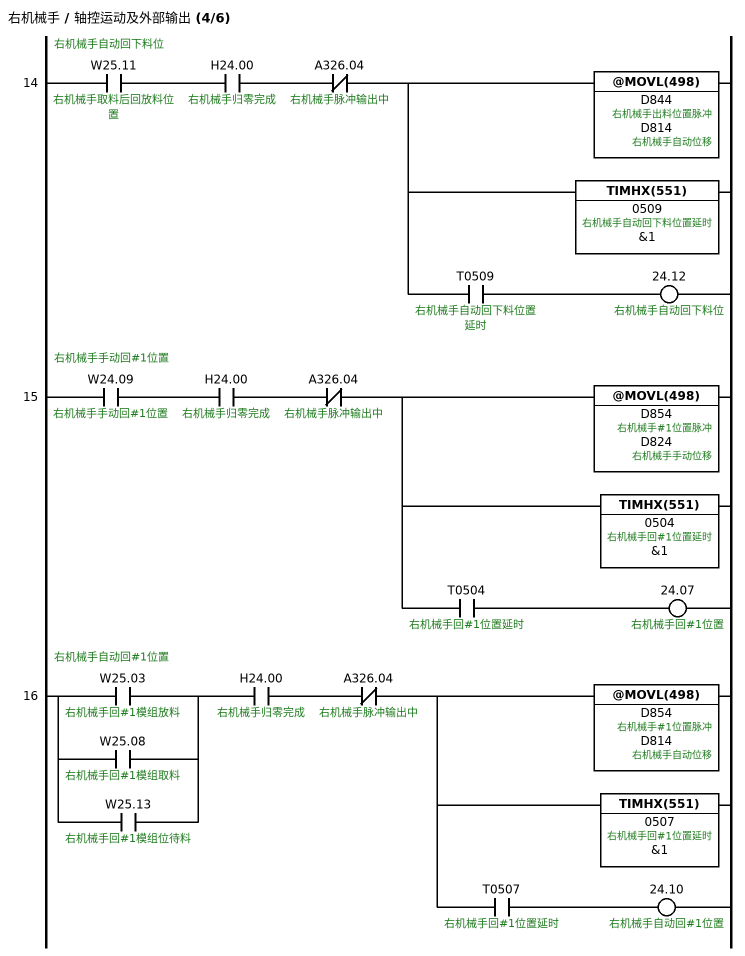
; [picture p185: 右机械手 / 轴控运动及外部输出, rungs 14-16]
; rung 14: 右机械手自动回下料位
LD W25.11  ; 右机械手取料后回放料位置
AND H24.00  ; 右机械手归零完成
ANDNOT A326.04  ; 右机械手脉冲输出中
@MOVL(498) D844 D814  ; 右机械手出料位置脉冲, 右机械手自动位移
TIMHX(551) 0509 &1  ; 右机械手自动回下料位置延时
AND T0509  ; 右机械手自动回下料位置延时
OUT 24.12  ; 右机械手自动回下料位
; rung 15: 右机械手手动回#1位置
LD W24.09  ; 右机械手手动回#1位置
AND H24.00  ; 右机械手归零完成
ANDNOT A326.04  ; 右机械手脉冲输出中
@MOVL(498) D854 D824  ; 右机械手#1位置脉冲, 右机械手手动位移
TIMHX(551) 0504 &1  ; 右机械手回#1位置延时
AND T0504  ; 右机械手回#1位置延时
OUT 24.07  ; 右机械手回#1位置
; rung 16: 右机械手自动回#1位置
LD W25.03  ; 右机械手回#1模组放料
OR W25.08  ; 右机械手回#1模组取料
OR W25.13  ; 右机械手回#1模组位待料
AND H24.00  ; 右机械手归零完成
ANDNOT A326.04  ; 右机械手脉冲输出中
@MOVL(498) D854 D814  ; 右机械手#1位置脉冲, 右机械手自动位移
TIMHX(551) 0507 &1  ; 右机械手回#1位置延时
AND T0507  ; 右机械手回#1位置延时
OUT 24.10  ; 右机械手自动回#1位置

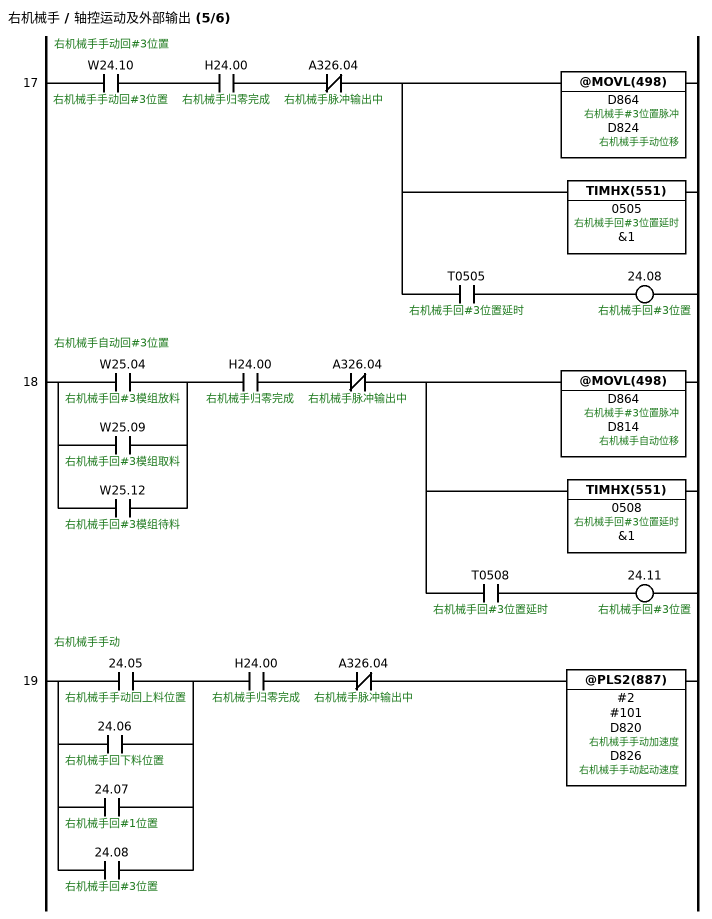
; rung 17: 右机械手手动回#3位置
LD W24.10  ; 右机械手手动回#3位置
AND H24.00  ; 右机械手归零完成
ANDNOT A326.04  ; 右机械手脉冲输出中
@MOVL(498) D864 D824  ; 右机械手#3位置脉冲, 右机械手手动位移
TIMHX(551) 0505 &1  ; 右机械手回#3位置延时
AND T0505  ; 右机械手回#3位置延时
OUT 24.08  ; 右机械手回#3位置
; rung 18: 右机械手自动回#3位置
LD W25.04  ; 右机械手回#3模组放料
OR W25.09  ; 右机械手回#3模组取料
OR W25.12  ; 右机械手回#3模组待料
AND H24.00  ; 右机械手归零完成
ANDNOT A326.04  ; 右机械手脉冲输出中
@MOVL(498) D864 D814  ; 右机械手#3位置脉冲, 右机械手自动位移
TIMHX(551) 0508 &1  ; 右机械手回#3位置延时
AND T0508  ; 右机械手回#3位置延时
OUT 24.11  ; 右机械手回#3位置
; rung 19: 右机械手手动
LD 24.05  ; 右机械手手动回上料位置
OR 24.06  ; 右机械手回下料位置
OR 24.07  ; 右机械手回#1位置
OR 24.08  ; 右机械手回#3位置
AND H24.00  ; 右机械手归零完成
ANDNOT A326.04  ; 右机械手脉冲输出中
@PLS2(887) #2 #101 D820 D826  ; 右机械手手动加速度, 右机械手手动起动速度

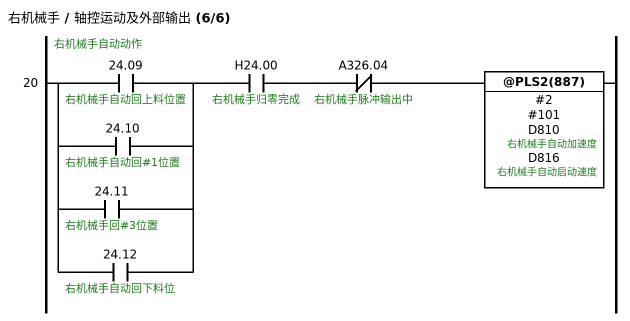
; rung 20: 右机械手自动动作
LD 24.09  ; 右机械手自动回上料位置
OR 24.10  ; 右机械手自动回#1位置
OR 24.11  ; 右机械手回#3位置
OR 24.12  ; 右机械手自动回下料位
AND H24.00  ; 右机械手归零完成
ANDNOT A326.04  ; 右机械手脉冲输出中
@PLS2(887) #2 #101 D810 D816  ; 右机械手自动加速度, 右机械手自动启动速度

### Section 自动报警

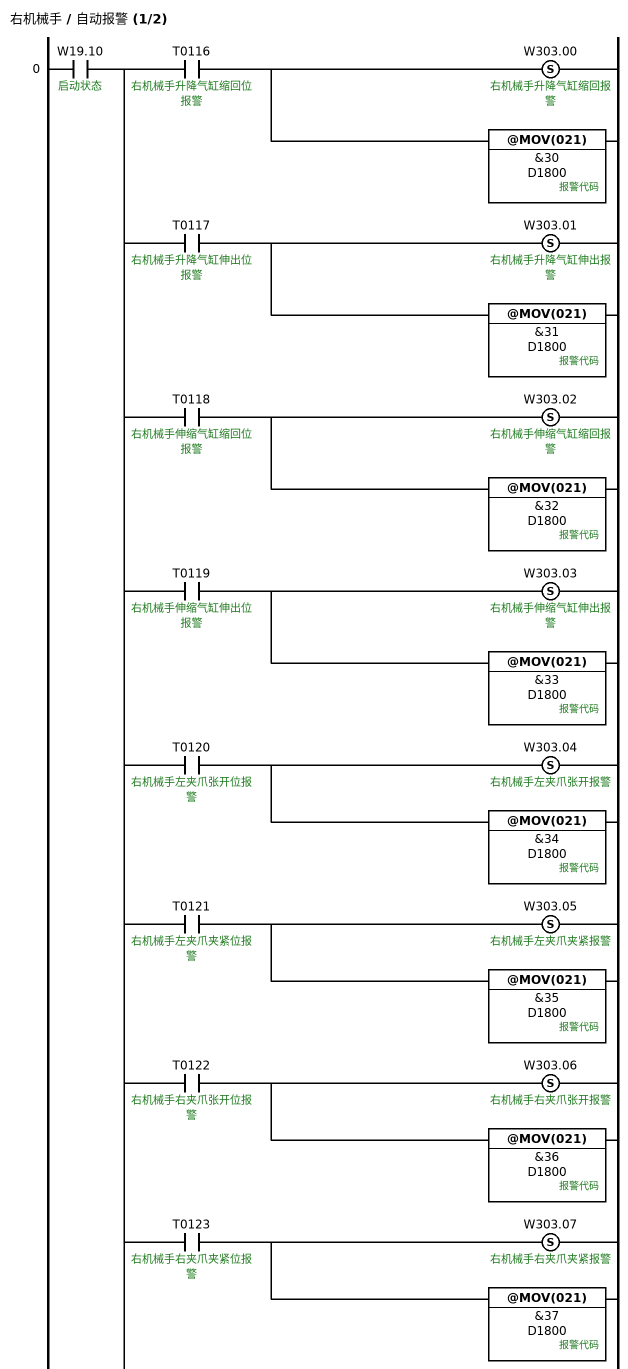

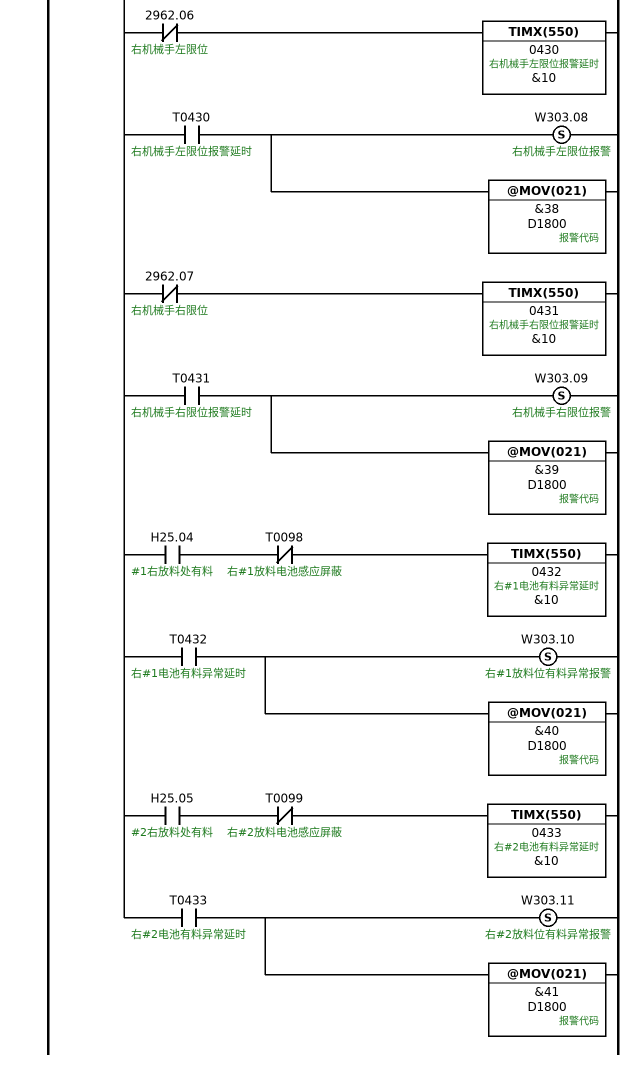
; rung 0
LD W19.10  ; 启动状态
OUT TR0
AND T0116  ; 右机械手升降气缸缩回位报警
SET W303.00  ; 右机械手升降气缸缩回报警
@MOV(021) &30 D1800  ; 报警代码
LD TR0
AND T0117  ; 右机械手升降气缸伸出位报警
SET W303.01  ; 右机械手升降气缸伸出报警
@MOV(021) &31 D1800  ; 报警代码
LD TR0
AND T0118  ; 右机械手伸缩气缸缩回位报警
SET W303.02  ; 右机械手伸缩气缸缩回报警
@MOV(021) &32 D1800  ; 报警代码
LD TR0
AND T0119  ; 右机械手伸缩气缸伸出位报警
SET W303.03  ; 右机械手伸缩气缸伸出报警
@MOV(021) &33 D1800  ; 报警代码
LD TR0
AND T0120  ; 右机械手左夹爪张开位报警
SET W303.04  ; 右机械手左夹爪张开报警
@MOV(021) &34 D1800  ; 报警代码
LD TR0
AND T0121  ; 右机械手左夹爪夹紧位报警
SET W303.05  ; 右机械手左夹爪夹紧报警
@MOV(021) &35 D1800  ; 报警代码
LD TR0
AND T0122  ; 右机械手右夹爪张开位报警
SET W303.06  ; 右机械手右夹爪张开报警
@MOV(021) &36 D1800  ; 报警代码
LD TR0
AND T0123  ; 右机械手右夹爪夹紧位报警
SET W303.07  ; 右机械手右夹爪夹紧报警
@MOV(021) &37 D1800  ; 报警代码
LD TR0
ANDNOT 2962.06  ; 右机械手左限位
TIMX(550) 0430 &10  ; 右机械手左限位报警延时
LD TR0
AND T0430  ; 右机械手左限位报警延时
SET W303.08  ; 右机械手左限位报警
@MOV(021) &38 D1800  ; 报警代码
LD TR0
ANDNOT 2962.07  ; 右机械手右限位
TIMX(550) 0431 &10  ; 右机械手右限位报警延时
LD TR0
AND T0431  ; 右机械手右限位报警延时
SET W303.09  ; 右机械手右限位报警
@MOV(021) &39 D1800  ; 报警代码
LD TR0
AND H25.04  ; #1右放料处有料
ANDNOT T0098  ; 右#1放料电池感应屏蔽
TIMX(550) 0432 &10  ; 右#1电池有料异常延时
LD TR0
AND T0432  ; 右#1电池有料异常延时
SET W303.10  ; 右#1放料位有料异常报警
@MOV(021) &40 D1800  ; 报警代码
LD TR0
AND H25.05  ; #2右放料处有料
ANDNOT T0099  ; 右#2放料电池感应屏蔽
TIMX(550) 0433 &10  ; 右#2电池有料异常延时
LD TR0
AND T0433  ; 右#2电池有料异常延时
SET W303.11  ; 右#2放料位有料异常报警
@MOV(021) &41 D1800  ; 报警代码

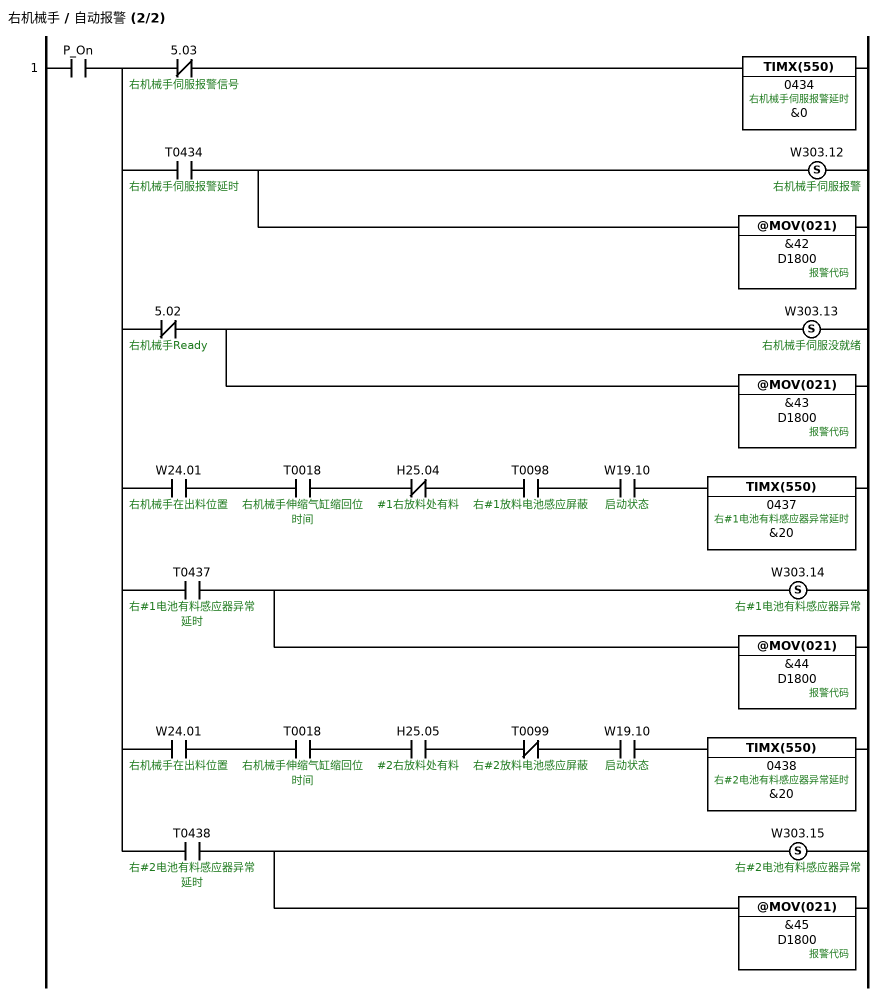
; rung 1
LD P_On
OUT TR0
ANDNOT 5.03  ; 右机械手伺服报警信号
TIMX(550) 0434 &0  ; 右机械手伺服报警延时
LD TR0
AND T0434  ; 右机械手伺服报警延时
SET W303.12  ; 右机械手伺服报警
@MOV(021) &42 D1800  ; 报警代码
LD TR0
ANDNOT 5.02  ; 右机械手Ready
SET W303.13  ; 右机械手伺服没就绪
@MOV(021) &43 D1800  ; 报警代码
LD TR0
AND W24.01  ; 右机械手在出料位置
AND T0018  ; 右机械手伸缩气缸缩回位时间
ANDNOT H25.04  ; #1右放料处有料
AND T0098  ; 右#1放料电池感应屏蔽
AND W19.10  ; 启动状态
TIMX(550) 0437 &20  ; 右#1电池有料感应器异常延时
LD TR0
AND T0437  ; 右#1电池有料感应器异常延时
SET W303.14  ; 右#1电池有料感应器异常
@MOV(021) &44 D1800  ; 报警代码
LD TR0
AND W24.01  ; 右机械手在出料位置
AND T0018  ; 右机械手伸缩气缸缩回位时间
AND H25.05  ; #2右放料处有料
ANDNOT T0099  ; 右#2放料电池感应屏蔽
AND W19.10  ; 启动状态
TIMX(550) 0438 &20  ; 右#2电池有料感应器异常延时
LD TR0
AND T0438  ; 右#2电池有料感应器异常延时
SET W303.15  ; 右#2电池有料感应器异常
@MOV(021) &45 D1800  ; 报警代码

### Section 右机械手复位

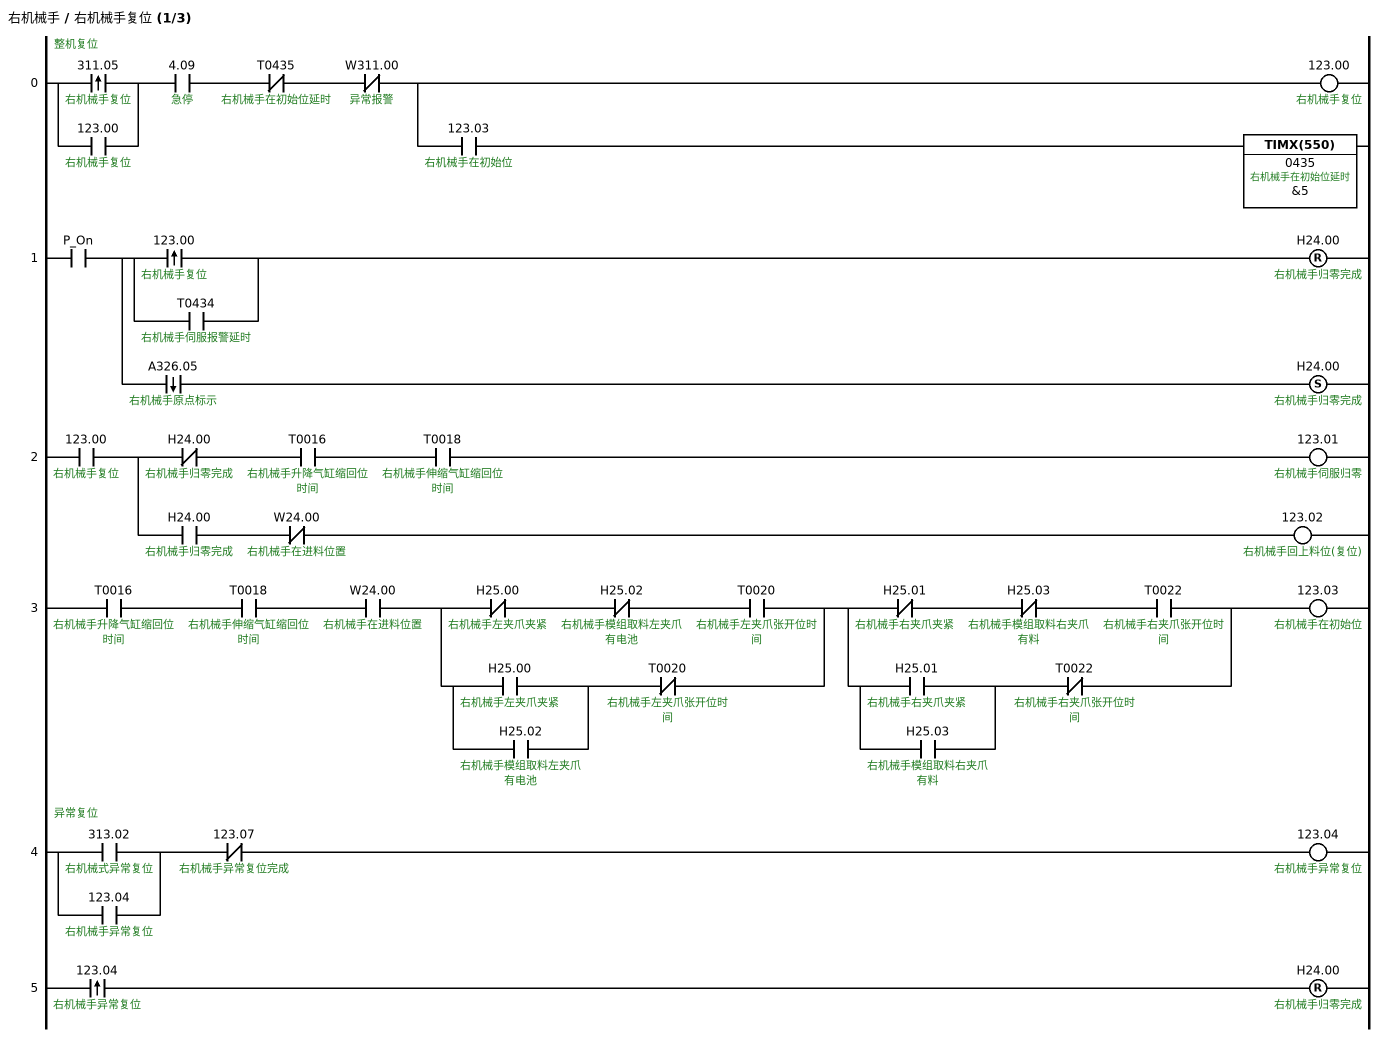
; rung 0: 整机复位
@LD 311.05  ; 右机械手复位
OR 123.00  ; 右机械手复位
AND 4.09  ; 急停
ANDNOT T0435  ; 右机械手在初始位延时
ANDNOT W311.00  ; 异常报警
OUT 123.00  ; 右机械手复位
AND 123.03  ; 右机械手在初始位
TIMX(550) 0435 &5  ; 右机械手在初始位延时
; rung 1
LD P_On
OUT TR0
@LD 123.00  ; 右机械手复位
OR T0434  ; 右机械手伺服报警延时
ANDLD
RSET H24.00  ; 右机械手归零完成
LD TR0
%AND A326.05  ; 右机械手原点标示
SET H24.00  ; 右机械手归零完成
; rung 2
LD 123.00  ; 右机械手复位
OUT TR0
ANDNOT H24.00  ; 右机械手归零完成
AND T0016  ; 右机械手升降气缸缩回位时间
AND T0018  ; 右机械手伸缩气缸缩回位时间
OUT 123.01  ; 右机械手伺服归零
LD TR0
AND H24.00  ; 右机械手归零完成
ANDNOT W24.00  ; 右机械手在进料位置
OUT 123.02  ; 右机械手回上料位(复位)
; rung 3
LD T0016  ; 右机械手升降气缸缩回位时间
AND T0018  ; 右机械手伸缩气缸缩回位时间
AND W24.00  ; 右机械手在进料位置
LDNOT H25.00  ; 右机械手左夹爪夹紧
ANDNOT H25.02  ; 右机械手模组取料左夹爪有电池
AND T0020  ; 右机械手左夹爪张开位时间
LD H25.00  ; 右机械手左夹爪夹紧
OR H25.02  ; 右机械手模组取料左夹爪有电池
ANDNOT T0020  ; 右机械手左夹爪张开位时间
ORLD
ANDLD
LDNOT H25.01  ; 右机械手右夹爪夹紧
ANDNOT H25.03  ; 右机械手模组取料右夹爪有料
AND T0022  ; 右机械手右夹爪张开位时间
LD H25.01  ; 右机械手右夹爪夹紧
OR H25.03  ; 右机械手模组取料右夹爪有料
ANDNOT T0022  ; 右机械手右夹爪张开位时间
ORLD
ANDLD
OUT 123.03  ; 右机械手在初始位
; rung 4: 异常复位
LD 313.02  ; 右机械式异常复位
OR 123.04  ; 右机械手异常复位
ANDNOT 123.07  ; 右机械手异常复位完成
OUT 123.04  ; 右机械手异常复位
; rung 5
@LD 123.04  ; 右机械手异常复位
RSET H24.00  ; 右机械手归零完成

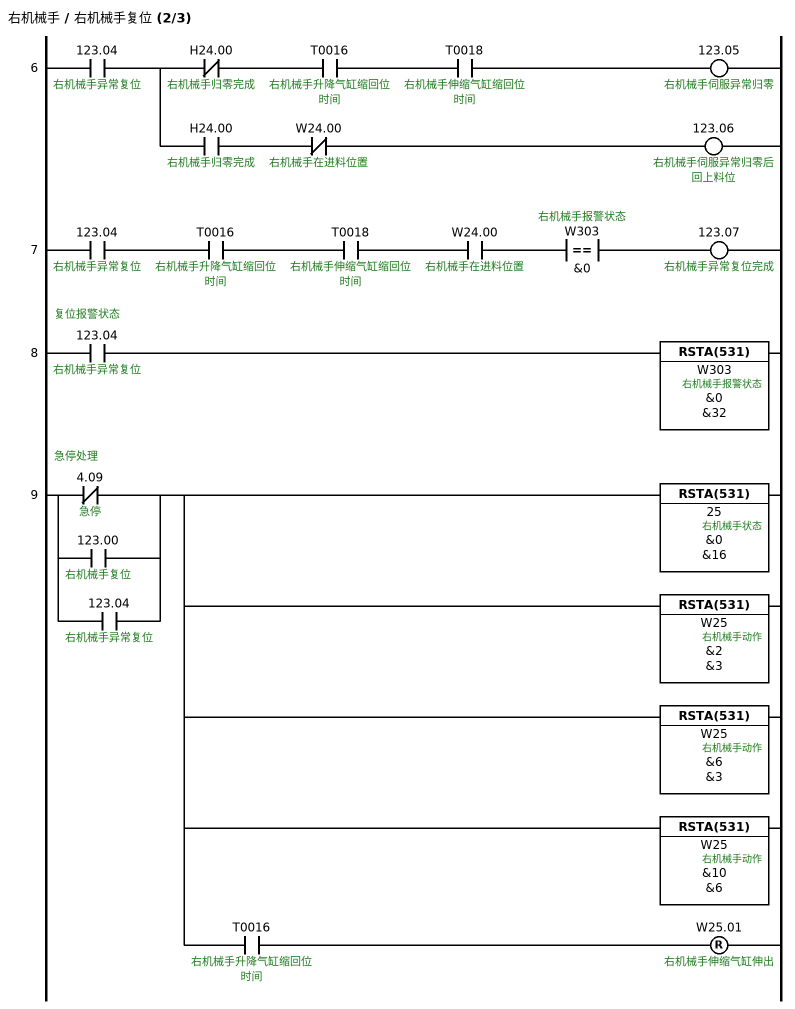
; rung 6
LD 123.04  ; 右机械手异常复位
OUT TR0
ANDNOT H24.00  ; 右机械手归零完成
AND T0016  ; 右机械手升降气缸缩回位时间
AND T0018  ; 右机械手伸缩气缸缩回位时间
OUT 123.05  ; 右机械手伺服异常归零
LD TR0
AND H24.00  ; 右机械手归零完成
ANDNOT W24.00  ; 右机械手在进料位置
OUT 123.06  ; 右机械手伺服异常归零后回上料位
; rung 7
LD 123.04  ; 右机械手异常复位
AND T0016  ; 右机械手升降气缸缩回位时间
AND T0018  ; 右机械手伸缩气缸缩回位时间
AND W24.00  ; 右机械手在进料位置
AND=L(301) W303 &0  ; 右机械手报警状态
OUT 123.07  ; 右机械手异常复位完成
; rung 8: 复位报警状态
LD 123.04  ; 右机械手异常复位
RSTA(531) W303 &0 &32  ; 右机械手报警状态
; rung 9: 急停处理
LDNOT 4.09  ; 急停
OR 123.00  ; 右机械手复位
OR 123.04  ; 右机械手异常复位
RSTA(531) 25 &0 &16  ; 右机械手状态
RSTA(531) W25 &2 &3  ; 右机械手动作
RSTA(531) W25 &6 &3  ; 右机械手动作
RSTA(531) W25 &10 &6  ; 右机械手动作
AND T0016  ; 右机械手升降气缸缩回位时间
RSET W25.01  ; 右机械手伸缩气缸伸出

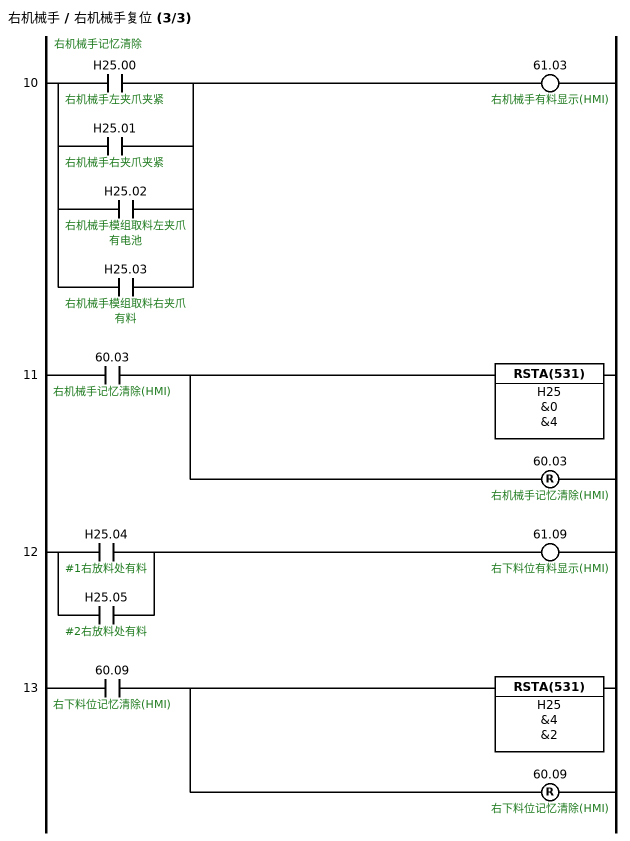
; rung 10: 右机械手记忆清除
LD H25.00  ; 右机械手左夹爪夹紧
OR H25.01  ; 右机械手右夹爪夹紧
OR H25.02  ; 右机械手模组取料左夹爪有电池
OR H25.03  ; 右机械手模组取料右夹爪有料
OUT 61.03  ; 右机械手有料显示(HMI)
; rung 11
LD 60.03  ; 右机械手记忆清除(HMI)
RSTA(531) H25 &0 &4
RSET 60.03  ; 右机械手记忆清除(HMI)
; rung 12
LD H25.04  ; #1右放料处有料
OR H25.05  ; #2右放料处有料
OUT 61.09  ; 右下料位有料显示(HMI)
; rung 13
LD 60.09  ; 右下料位记忆清除(HMI)
RSTA(531) H25 &4 &2
RSET 60.09  ; 右下料位记忆清除(HMI)

### Section END
; rung 0
END(001)

## Program 模组 (cyclic task 6)
Local symbols
P_off BOOL  ; 常段标志
w BOOL

### Section 模组_1手动

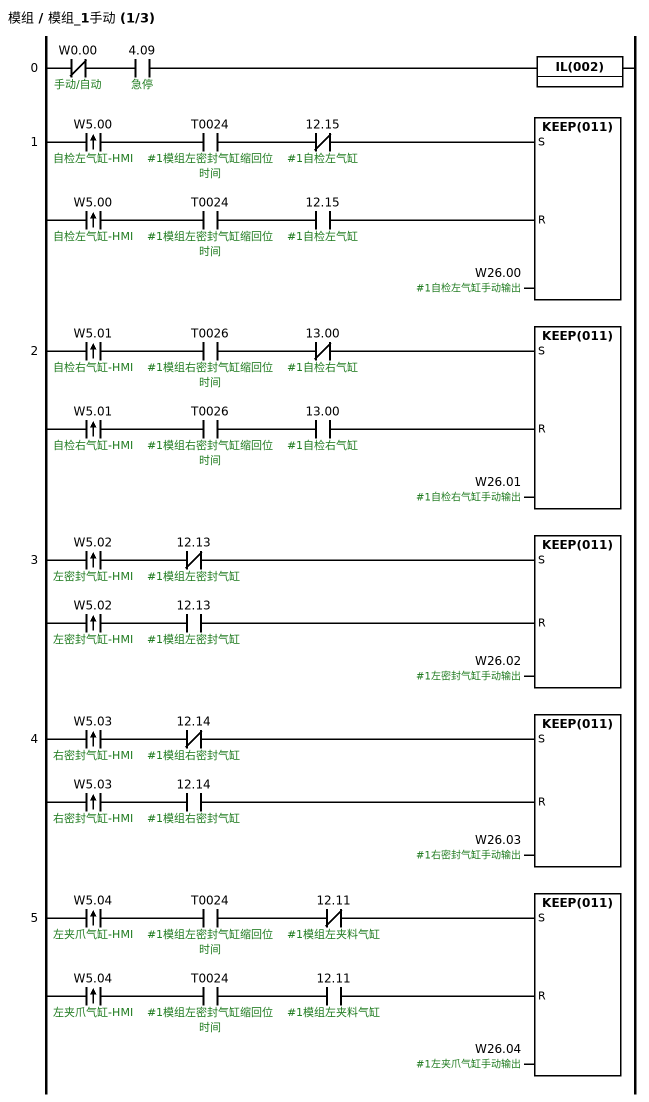
; rung 0
LDNOT W0.00  ; 手动/自动
AND 4.09  ; 急停
IL(002)
; rung 1
@LD W5.00  ; 自检左气缸-HMI
AND T0024  ; #1模组左密封气缸缩回位时间
ANDNOT 12.15  ; #1自检左气缸
@LD W5.00  ; 自检左气缸-HMI
AND T0024  ; #1模组左密封气缸缩回位时间
AND 12.15  ; #1自检左气缸
KEEP(011) W26.00  ; #1自检左气缸手动输出
; rung 2
@LD W5.01  ; 自检右气缸-HMI
AND T0026  ; #1模组右密封气缸缩回位时间
ANDNOT 13.00  ; #1自检右气缸
@LD W5.01  ; 自检右气缸-HMI
AND T0026  ; #1模组右密封气缸缩回位时间
AND 13.00  ; #1自检右气缸
KEEP(011) W26.01  ; #1自检右气缸手动输出
; rung 3
@LD W5.02  ; 左密封气缸-HMI
ANDNOT 12.13  ; #1模组左密封气缸
@LD W5.02  ; 左密封气缸-HMI
AND 12.13  ; #1模组左密封气缸
KEEP(011) W26.02  ; #1左密封气缸手动输出
; rung 4
@LD W5.03  ; 右密封气缸-HMI
ANDNOT 12.14  ; #1模组右密封气缸
@LD W5.03  ; 右密封气缸-HMI
AND 12.14  ; #1模组右密封气缸
KEEP(011) W26.03  ; #1右密封气缸手动输出
; rung 5
@LD W5.04  ; 左夹爪气缸-HMI
AND T0024  ; #1模组左密封气缸缩回位时间
ANDNOT 12.11  ; #1模组左夹料气缸
@LD W5.04  ; 左夹爪气缸-HMI
AND T0024  ; #1模组左密封气缸缩回位时间
AND 12.11  ; #1模组左夹料气缸
KEEP(011) W26.04  ; #1左夹爪气缸手动输出

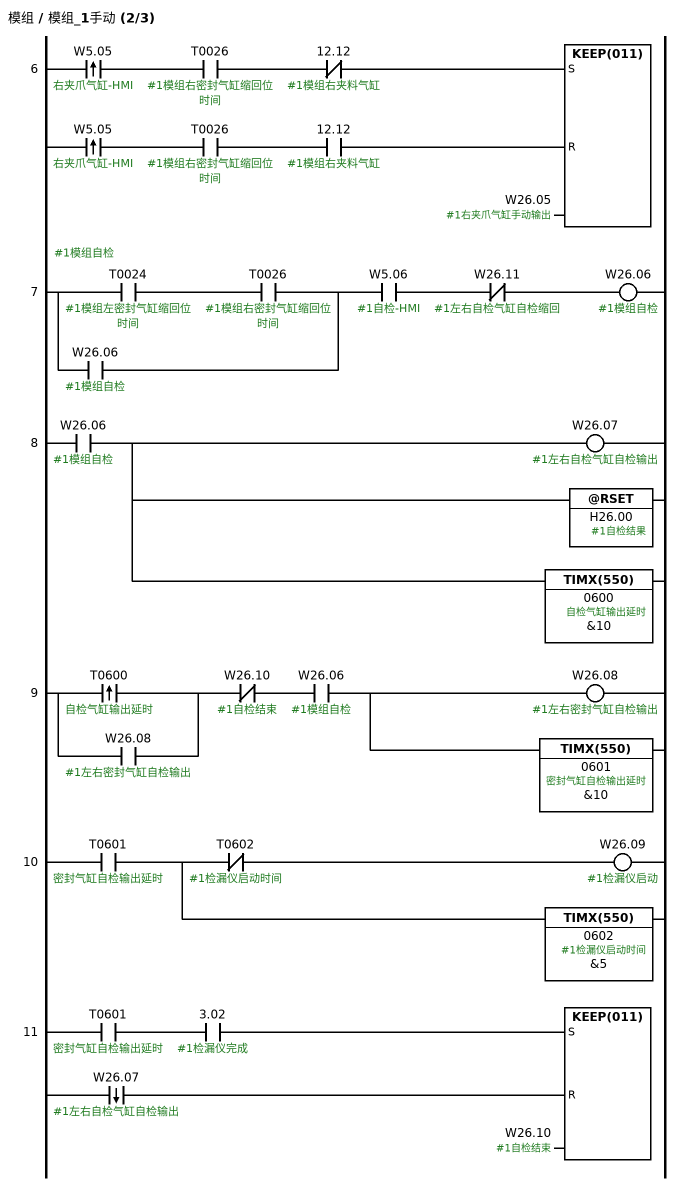
; rung 6
@LD W5.05  ; 右夹爪气缸-HMI
AND T0026  ; #1模组右密封气缸缩回位时间
ANDNOT 12.12  ; #1模组右夹料气缸
@LD W5.05  ; 右夹爪气缸-HMI
AND T0026  ; #1模组右密封气缸缩回位时间
AND 12.12  ; #1模组右夹料气缸
KEEP(011) W26.05  ; #1右夹爪气缸手动输出
; rung 7: #1模组自检
LD T0024  ; #1模组左密封气缸缩回位时间
AND T0026  ; #1模组右密封气缸缩回位时间
OR W26.06  ; #1模组自检
AND W5.06  ; #1自检-HMI
ANDNOT W26.11  ; #1左右自检气缸自检缩回
OUT W26.06  ; #1模组自检
; rung 8
LD W26.06  ; #1模组自检
OUT W26.07  ; #1左右自检气缸自检输出
@RSET H26.00  ; #1自检结果
TIMX(550) 0600 &10  ; 自检气缸输出延时
; rung 9
@LD T0600  ; 自检气缸输出延时
OR W26.08  ; #1左右密封气缸自检输出
ANDNOT W26.10  ; #1自检结束
AND W26.06  ; #1模组自检
OUT W26.08  ; #1左右密封气缸自检输出
TIMX(550) 0601 &10  ; 密封气缸自检输出延时
; rung 10
LD T0601  ; 密封气缸自检输出延时
OUT TR0
ANDNOT T0602  ; #1检漏仪启动时间
OUT W26.09  ; #1检漏仪启动
LD TR0
TIMX(550) 0602 &5  ; #1检漏仪启动时间
; rung 11
LD T0601  ; 密封气缸自检输出延时
AND 3.02  ; #1检漏仪完成
%LD W26.07  ; #1左右自检气缸自检输出
KEEP(011) W26.10  ; #1自检结束

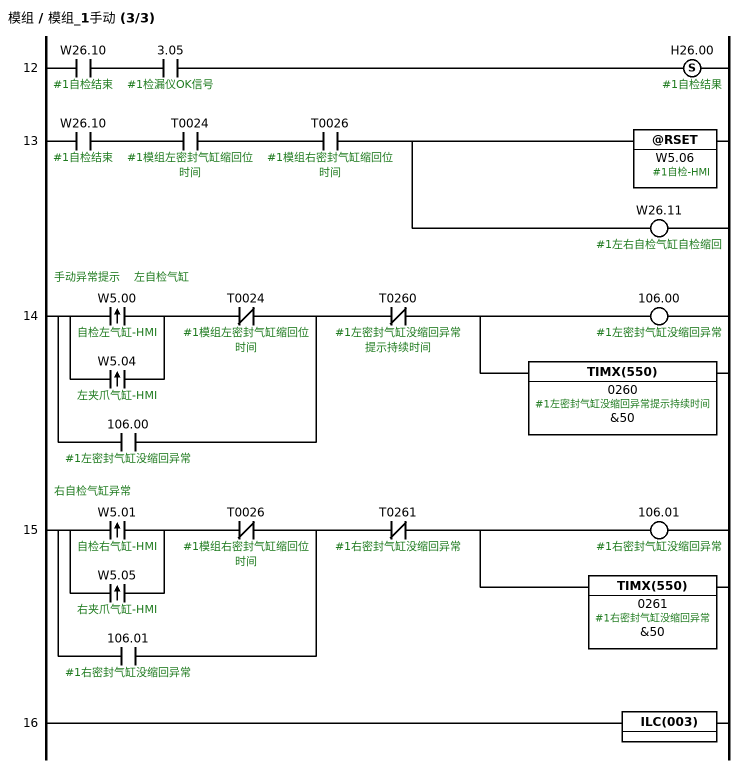
; rung 12
LD W26.10  ; #1自检结束
AND 3.05  ; #1检漏仪OK信号
SET H26.00  ; #1自检结果
; rung 13
LD W26.10  ; #1自检结束
AND T0024  ; #1模组左密封气缸缩回位时间
AND T0026  ; #1模组右密封气缸缩回位时间
@RSET W5.06  ; #1自检-HMI
OUT W26.11  ; #1左右自检气缸自检缩回
; rung 14: 手动异常提示    左自检气缸
@LD W5.00  ; 自检左气缸-HMI
@OR W5.04  ; 左夹爪气缸-HMI
ANDNOT T0024  ; #1模组左密封气缸缩回位时间
OR 106.00  ; #1左密封气缸没缩回异常
ANDNOT T0260  ; #1左密封气缸没缩回异常提示持续时间
OUT 106.00  ; #1左密封气缸没缩回异常
TIMX(550) 0260 &50  ; #1左密封气缸没缩回异常提示持续时间
; rung 15: 右自检气缸异常
@LD W5.01  ; 自检右气缸-HMI
@OR W5.05  ; 右夹爪气缸-HMI
ANDNOT T0026  ; #1模组右密封气缸缩回位时间
OR 106.01  ; #1右密封气缸没缩回异常
ANDNOT T0261  ; #1右密封气缸没缩回异常
OUT 106.01  ; #1右密封气缸没缩回异常
TIMX(550) 0261 &50  ; #1右密封气缸没缩回异常
; rung 16
ILC(003)

### Section 模组_2手动

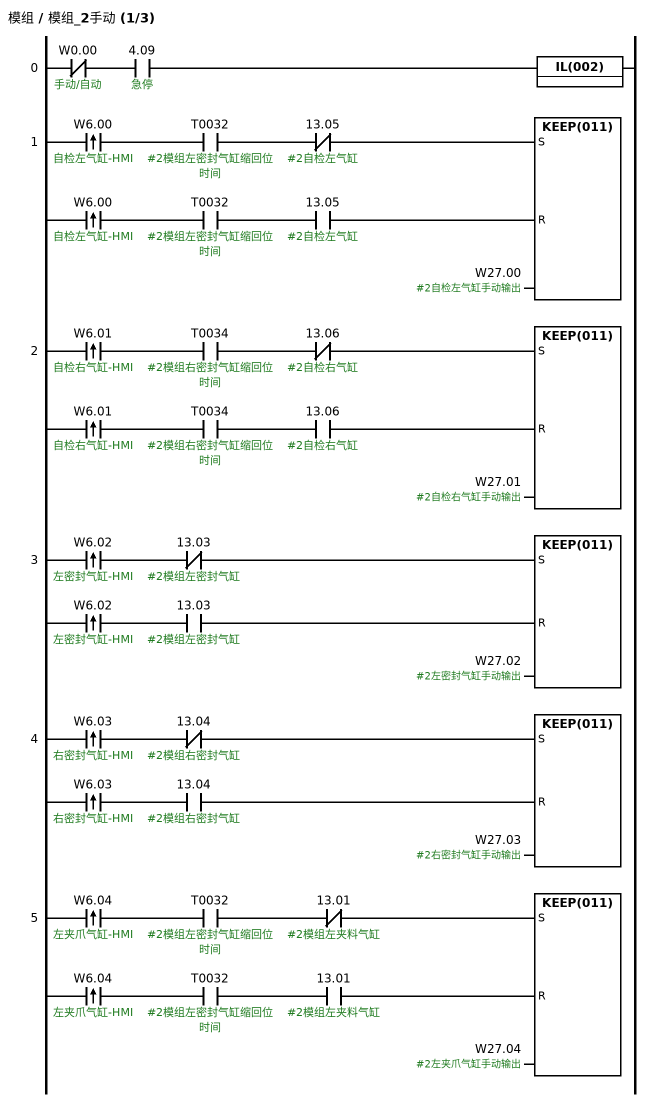
; rung 0
LDNOT W0.00  ; 手动/自动
AND 4.09  ; 急停
IL(002)
; rung 1
@LD W6.00  ; 自检左气缸-HMI
AND T0032  ; #2模组左密封气缸缩回位时间
ANDNOT 13.05  ; #2自检左气缸
@LD W6.00  ; 自检左气缸-HMI
AND T0032  ; #2模组左密封气缸缩回位时间
AND 13.05  ; #2自检左气缸
KEEP(011) W27.00  ; #2自检左气缸手动输出
; rung 2
@LD W6.01  ; 自检右气缸-HMI
AND T0034  ; #2模组右密封气缸缩回位时间
ANDNOT 13.06  ; #2自检右气缸
@LD W6.01  ; 自检右气缸-HMI
AND T0034  ; #2模组右密封气缸缩回位时间
AND 13.06  ; #2自检右气缸
KEEP(011) W27.01  ; #2自检右气缸手动输出
; rung 3
@LD W6.02  ; 左密封气缸-HMI
ANDNOT 13.03  ; #2模组左密封气缸
@LD W6.02  ; 左密封气缸-HMI
AND 13.03  ; #2模组左密封气缸
KEEP(011) W27.02  ; #2左密封气缸手动输出
; rung 4
@LD W6.03  ; 右密封气缸-HMI
ANDNOT 13.04  ; #2模组右密封气缸
@LD W6.03  ; 右密封气缸-HMI
AND 13.04  ; #2模组右密封气缸
KEEP(011) W27.03  ; #2右密封气缸手动输出
; rung 5
@LD W6.04  ; 左夹爪气缸-HMI
AND T0032  ; #2模组左密封气缸缩回位时间
ANDNOT 13.01  ; #2模组左夹料气缸
@LD W6.04  ; 左夹爪气缸-HMI
AND T0032  ; #2模组左密封气缸缩回位时间
AND 13.01  ; #2模组左夹料气缸
KEEP(011) W27.04  ; #2左夹爪气缸手动输出

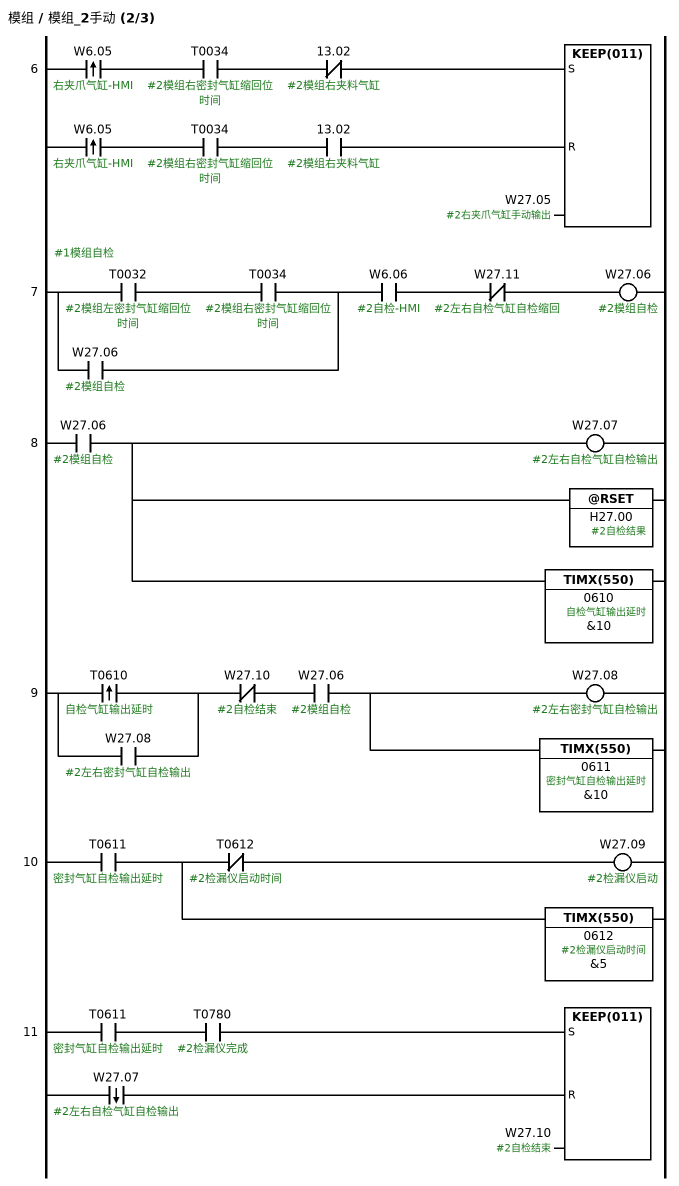
; rung 6
@LD W6.05  ; 右夹爪气缸-HMI
AND T0034  ; #2模组右密封气缸缩回位时间
ANDNOT 13.02  ; #2模组右夹料气缸
@LD W6.05  ; 右夹爪气缸-HMI
AND T0034  ; #2模组右密封气缸缩回位时间
AND 13.02  ; #2模组右夹料气缸
KEEP(011) W27.05  ; #2右夹爪气缸手动输出
; rung 7: #1模组自检
LD T0032  ; #2模组左密封气缸缩回位时间
AND T0034  ; #2模组右密封气缸缩回位时间
OR W27.06  ; #2模组自检
AND W6.06  ; #2自检-HMI
ANDNOT W27.11  ; #2左右自检气缸自检缩回
OUT W27.06  ; #2模组自检
; rung 8
LD W27.06  ; #2模组自检
OUT W27.07  ; #2左右自检气缸自检输出
@RSET H27.00  ; #2自检结果
TIMX(550) 0610 &10  ; 自检气缸输出延时
; rung 9
@LD T0610  ; 自检气缸输出延时
OR W27.08  ; #2左右密封气缸自检输出
ANDNOT W27.10  ; #2自检结束
AND W27.06  ; #2模组自检
OUT W27.08  ; #2左右密封气缸自检输出
TIMX(550) 0611 &10  ; 密封气缸自检输出延时
; rung 10
LD T0611  ; 密封气缸自检输出延时
OUT TR0
ANDNOT T0612  ; #2检漏仪启动时间
OUT W27.09  ; #2检漏仪启动
LD TR0
TIMX(550) 0612 &5  ; #2检漏仪启动时间
; rung 11
LD T0611  ; 密封气缸自检输出延时
AND T0780  ; #2检漏仪完成
%LD W27.07  ; #2左右自检气缸自检输出
KEEP(011) W27.10  ; #2自检结束

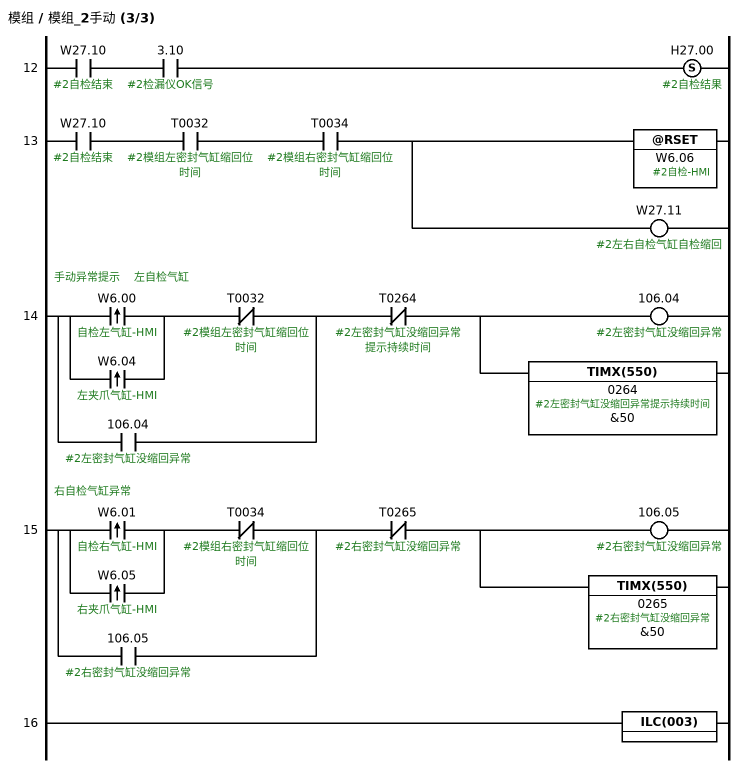
; rung 12
LD W27.10  ; #2自检结束
AND 3.10  ; #2检漏仪OK信号
SET H27.00  ; #2自检结果
; rung 13
LD W27.10  ; #2自检结束
AND T0032  ; #2模组左密封气缸缩回位时间
AND T0034  ; #2模组右密封气缸缩回位时间
@RSET W6.06  ; #2自检-HMI
OUT W27.11  ; #2左右自检气缸自检缩回
; rung 14: 手动异常提示    左自检气缸
@LD W6.00  ; 自检左气缸-HMI
@OR W6.04  ; 左夹爪气缸-HMI
ANDNOT T0032  ; #2模组左密封气缸缩回位时间
OR 106.04  ; #2左密封气缸没缩回异常
ANDNOT T0264  ; #2左密封气缸没缩回异常提示持续时间
OUT 106.04  ; #2左密封气缸没缩回异常
TIMX(550) 0264 &50  ; #2左密封气缸没缩回异常提示持续时间
; rung 15: 右自检气缸异常
@LD W6.01  ; 自检右气缸-HMI
@OR W6.05  ; 右夹爪气缸-HMI
ANDNOT T0034  ; #2模组右密封气缸缩回位时间
OR 106.05  ; #2右密封气缸没缩回异常
ANDNOT T0265  ; #2右密封气缸没缩回异常
OUT 106.05  ; #2右密封气缸没缩回异常
TIMX(550) 0265 &50  ; #2右密封气缸没缩回异常
; rung 16
ILC(003)

### Section 模组_3手动

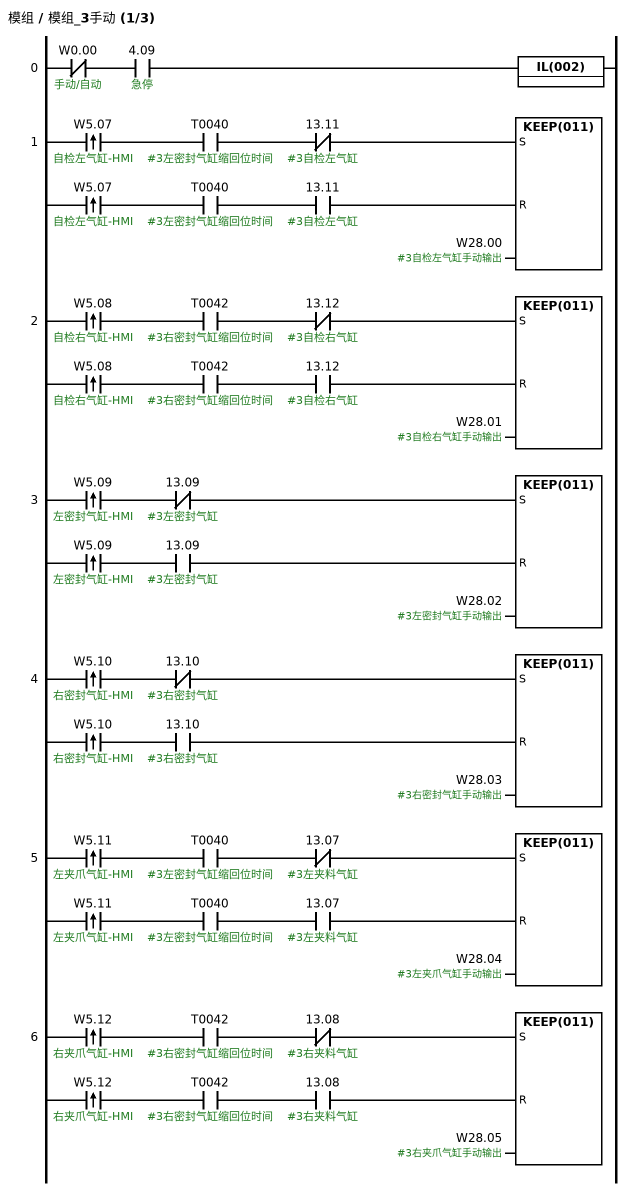
; rung 0
LDNOT W0.00  ; 手动/自动
AND 4.09  ; 急停
IL(002)
; rung 1
@LD W5.07  ; 自检左气缸-HMI
AND T0040  ; #3左密封气缸缩回位时间
ANDNOT 13.11  ; #3自检左气缸
@LD W5.07  ; 自检左气缸-HMI
AND T0040  ; #3左密封气缸缩回位时间
AND 13.11  ; #3自检左气缸
KEEP(011) W28.00  ; #3自检左气缸手动输出
; rung 2
@LD W5.08  ; 自检右气缸-HMI
AND T0042  ; #3右密封气缸缩回位时间
ANDNOT 13.12  ; #3自检右气缸
@LD W5.08  ; 自检右气缸-HMI
AND T0042  ; #3右密封气缸缩回位时间
AND 13.12  ; #3自检右气缸
KEEP(011) W28.01  ; #3自检右气缸手动输出
; rung 3
@LD W5.09  ; 左密封气缸-HMI
ANDNOT 13.09  ; #3左密封气缸
@LD W5.09  ; 左密封气缸-HMI
AND 13.09  ; #3左密封气缸
KEEP(011) W28.02  ; #3左密封气缸手动输出
; rung 4
@LD W5.10  ; 右密封气缸-HMI
ANDNOT 13.10  ; #3右密封气缸
@LD W5.10  ; 右密封气缸-HMI
AND 13.10  ; #3右密封气缸
KEEP(011) W28.03  ; #3右密封气缸手动输出
; rung 5
@LD W5.11  ; 左夹爪气缸-HMI
AND T0040  ; #3左密封气缸缩回位时间
ANDNOT 13.07  ; #3左夹料气缸
@LD W5.11  ; 左夹爪气缸-HMI
AND T0040  ; #3左密封气缸缩回位时间
AND 13.07  ; #3左夹料气缸
KEEP(011) W28.04  ; #3左夹爪气缸手动输出
; rung 6
@LD W5.12  ; 右夹爪气缸-HMI
AND T0042  ; #3右密封气缸缩回位时间
ANDNOT 13.08  ; #3右夹料气缸
@LD W5.12  ; 右夹爪气缸-HMI
AND T0042  ; #3右密封气缸缩回位时间
AND 13.08  ; #3右夹料气缸
KEEP(011) W28.05  ; #3右夹爪气缸手动输出

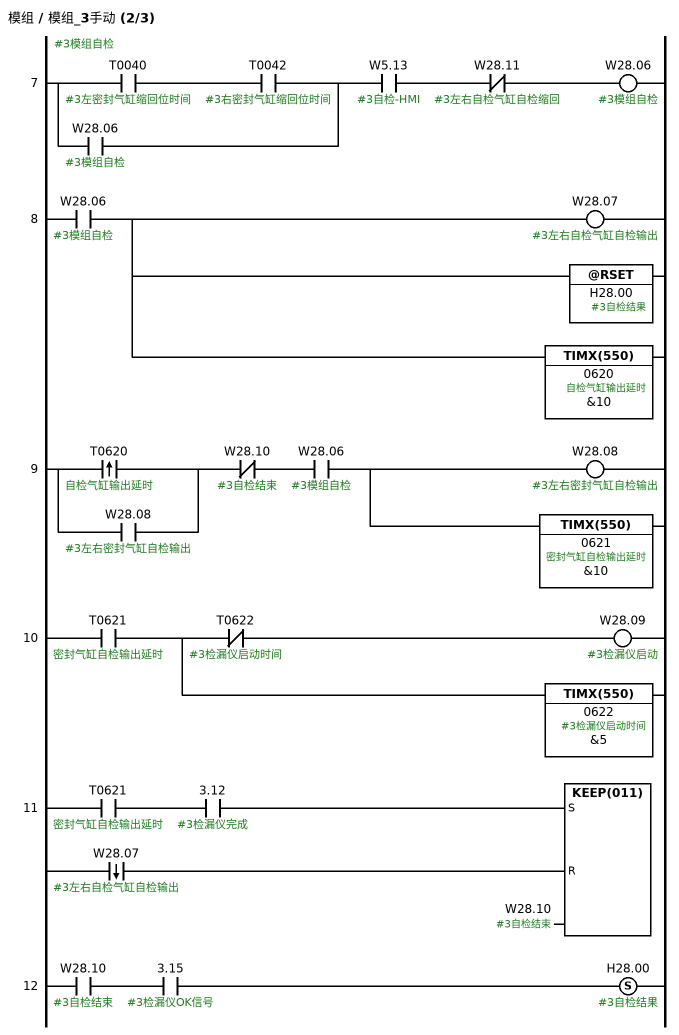
; rung 7: #3模组自检
LD T0040  ; #3左密封气缸缩回位时间
AND T0042  ; #3右密封气缸缩回位时间
OR W28.06  ; #3模组自检
AND W5.13  ; #3自检-HMI
ANDNOT W28.11  ; #3左右自检气缸自检缩回
OUT W28.06  ; #3模组自检
; rung 8
LD W28.06  ; #3模组自检
OUT W28.07  ; #3左右自检气缸自检输出
@RSET H28.00  ; #3自检结果
TIMX(550) 0620 &10  ; 自检气缸输出延时
; rung 9
@LD T0620  ; 自检气缸输出延时
OR W28.08  ; #3左右密封气缸自检输出
ANDNOT W28.10  ; #3自检结束
AND W28.06  ; #3模组自检
OUT W28.08  ; #3左右密封气缸自检输出
TIMX(550) 0621 &10  ; 密封气缸自检输出延时
; rung 10
LD T0621  ; 密封气缸自检输出延时
OUT TR0
ANDNOT T0622  ; #3检漏仪启动时间
OUT W28.09  ; #3检漏仪启动
LD TR0
TIMX(550) 0622 &5  ; #3检漏仪启动时间
; rung 11
LD T0621  ; 密封气缸自检输出延时
AND 3.12  ; #3检漏仪完成
%LD W28.07  ; #3左右自检气缸自检输出
KEEP(011) W28.10  ; #3自检结束
; rung 12
LD W28.10  ; #3自检结束
AND 3.15  ; #3检漏仪OK信号
SET H28.00  ; #3自检结果

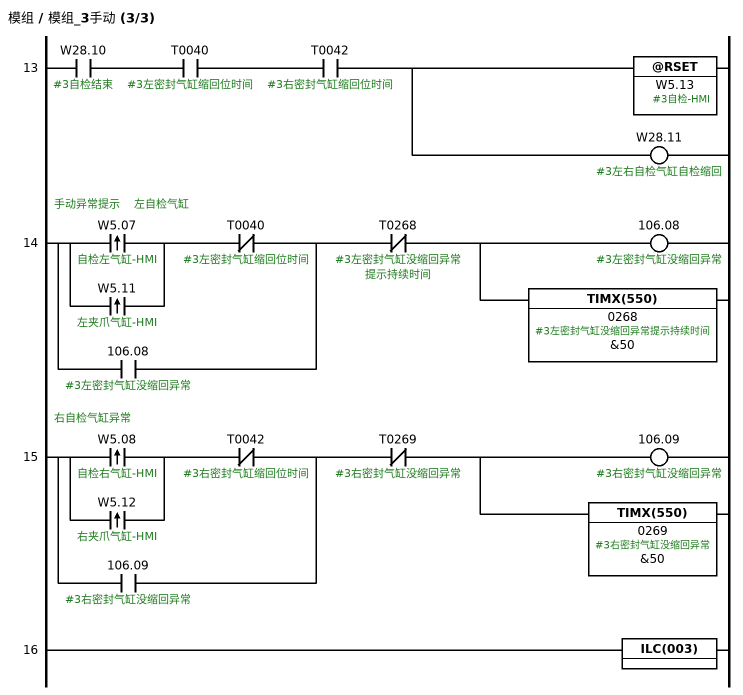
; rung 13
LD W28.10  ; #3自检结束
AND T0040  ; #3左密封气缸缩回位时间
AND T0042  ; #3右密封气缸缩回位时间
@RSET W5.13  ; #3自检-HMI
OUT W28.11  ; #3左右自检气缸自检缩回
; rung 14: 手动异常提示    左自检气缸
@LD W5.07  ; 自检左气缸-HMI
@OR W5.11  ; 左夹爪气缸-HMI
ANDNOT T0040  ; #3左密封气缸缩回位时间
OR 106.08  ; #3左密封气缸没缩回异常
ANDNOT T0268  ; #3左密封气缸没缩回异常提示持续时间
OUT 106.08  ; #3左密封气缸没缩回异常
TIMX(550) 0268 &50  ; #3左密封气缸没缩回异常提示持续时间
; rung 15: 右自检气缸异常
@LD W5.08  ; 自检右气缸-HMI
@OR W5.12  ; 右夹爪气缸-HMI
ANDNOT T0042  ; #3右密封气缸缩回位时间
OR 106.09  ; #3右密封气缸没缩回异常
ANDNOT T0269  ; #3右密封气缸没缩回异常
OUT 106.09  ; #3右密封气缸没缩回异常
TIMX(550) 0269 &50  ; #3右密封气缸没缩回异常
; rung 16
ILC(003)

### Section 模组_4手动

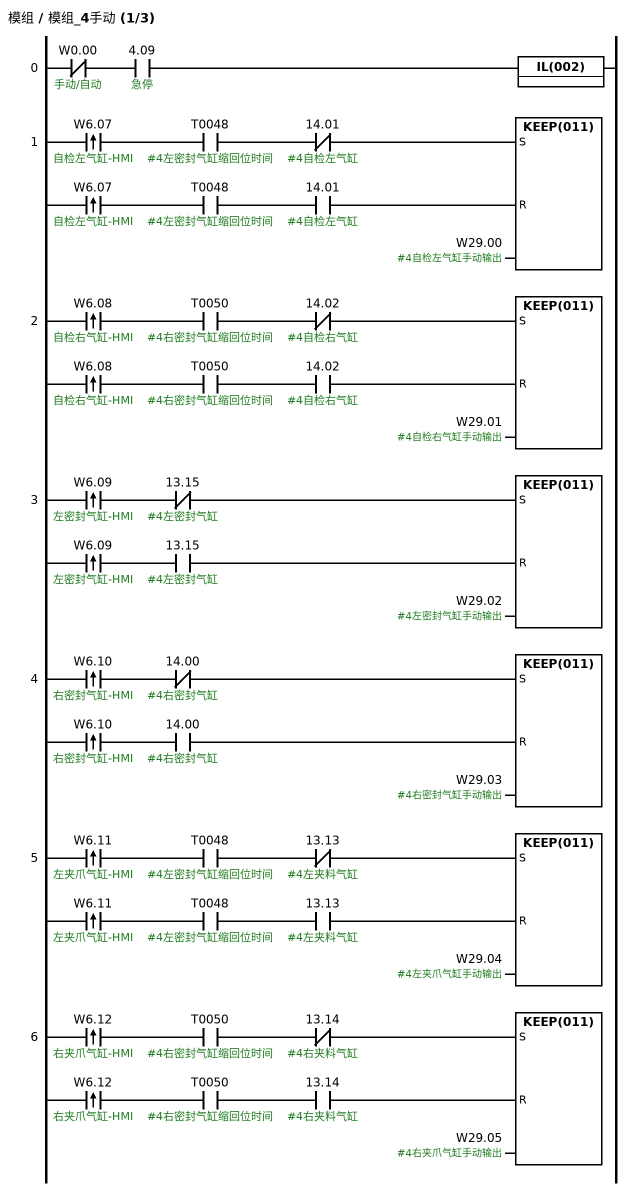
; rung 0
LDNOT W0.00  ; 手动/自动
AND 4.09  ; 急停
IL(002)
; rung 1
@LD W6.07  ; 自检左气缸-HMI
AND T0048  ; #4左密封气缸缩回位时间
ANDNOT 14.01  ; #4自检左气缸
@LD W6.07  ; 自检左气缸-HMI
AND T0048  ; #4左密封气缸缩回位时间
AND 14.01  ; #4自检左气缸
KEEP(011) W29.00  ; #4自检左气缸手动输出
; rung 2
@LD W6.08  ; 自检右气缸-HMI
AND T0050  ; #4右密封气缸缩回位时间
ANDNOT 14.02  ; #4自检右气缸
@LD W6.08  ; 自检右气缸-HMI
AND T0050  ; #4右密封气缸缩回位时间
AND 14.02  ; #4自检右气缸
KEEP(011) W29.01  ; #4自检右气缸手动输出
; rung 3
@LD W6.09  ; 左密封气缸-HMI
ANDNOT 13.15  ; #4左密封气缸
@LD W6.09  ; 左密封气缸-HMI
AND 13.15  ; #4左密封气缸
KEEP(011) W29.02  ; #4左密封气缸手动输出
; rung 4
@LD W6.10  ; 右密封气缸-HMI
ANDNOT 14.00  ; #4右密封气缸
@LD W6.10  ; 右密封气缸-HMI
AND 14.00  ; #4右密封气缸
KEEP(011) W29.03  ; #4右密封气缸手动输出
; rung 5
@LD W6.11  ; 左夹爪气缸-HMI
AND T0048  ; #4左密封气缸缩回位时间
ANDNOT 13.13  ; #4左夹料气缸
@LD W6.11  ; 左夹爪气缸-HMI
AND T0048  ; #4左密封气缸缩回位时间
AND 13.13  ; #4左夹料气缸
KEEP(011) W29.04  ; #4左夹爪气缸手动输出
; rung 6
@LD W6.12  ; 右夹爪气缸-HMI
AND T0050  ; #4右密封气缸缩回位时间
ANDNOT 13.14  ; #4右夹料气缸
@LD W6.12  ; 右夹爪气缸-HMI
AND T0050  ; #4右密封气缸缩回位时间
AND 13.14  ; #4右夹料气缸
KEEP(011) W29.05  ; #4右夹爪气缸手动输出

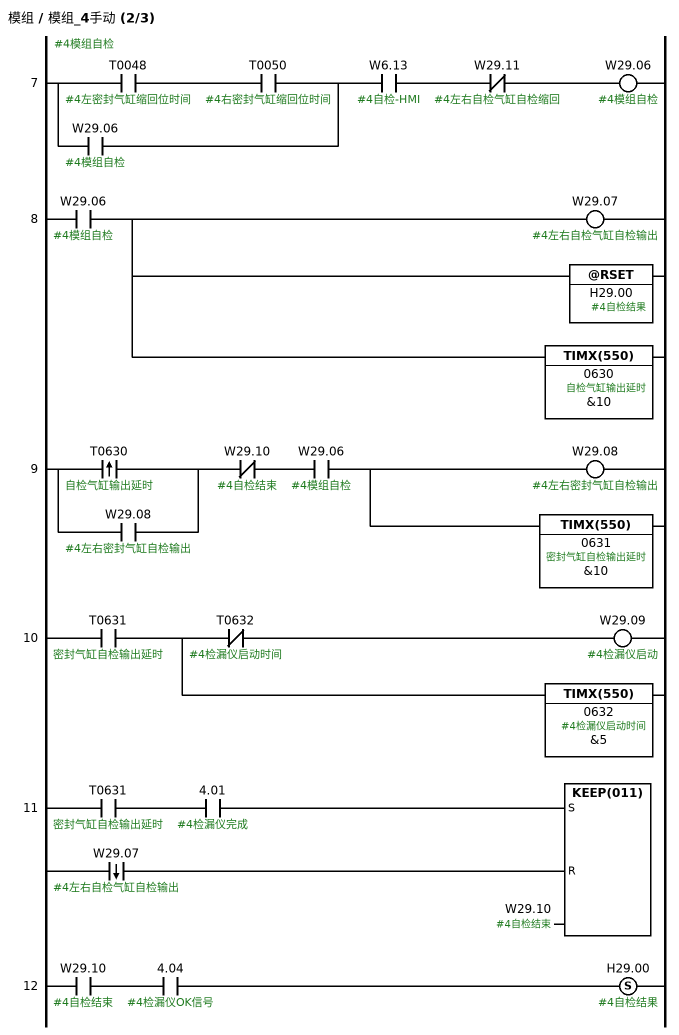
; rung 7: #4模组自检
LD T0048  ; #4左密封气缸缩回位时间
AND T0050  ; #4右密封气缸缩回位时间
OR W29.06  ; #4模组自检
AND W6.13  ; #4自检-HMI
ANDNOT W29.11  ; #4左右自检气缸自检缩回
OUT W29.06  ; #4模组自检
; rung 8
LD W29.06  ; #4模组自检
OUT W29.07  ; #4左右自检气缸自检输出
@RSET H29.00  ; #4自检结果
TIMX(550) 0630 &10  ; 自检气缸输出延时
; rung 9
@LD T0630  ; 自检气缸输出延时
OR W29.08  ; #4左右密封气缸自检输出
ANDNOT W29.10  ; #4自检结束
AND W29.06  ; #4模组自检
OUT W29.08  ; #4左右密封气缸自检输出
TIMX(550) 0631 &10  ; 密封气缸自检输出延时
; rung 10
LD T0631  ; 密封气缸自检输出延时
OUT TR0
ANDNOT T0632  ; #4检漏仪启动时间
OUT W29.09  ; #4检漏仪启动
LD TR0
TIMX(550) 0632 &5  ; #4检漏仪启动时间
; rung 11
LD T0631  ; 密封气缸自检输出延时
AND 4.01  ; #4检漏仪完成
%LD W29.07  ; #4左右自检气缸自检输出
KEEP(011) W29.10  ; #4自检结束
; rung 12
LD W29.10  ; #4自检结束
AND 4.04  ; #4检漏仪OK信号
SET H29.00  ; #4自检结果

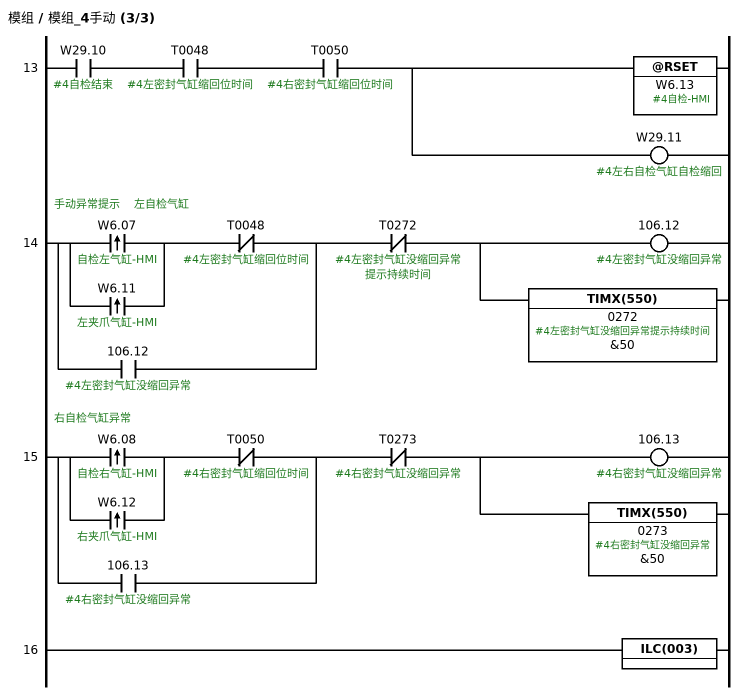
; rung 13
LD W29.10  ; #4自检结束
AND T0048  ; #4左密封气缸缩回位时间
AND T0050  ; #4右密封气缸缩回位时间
@RSET W6.13  ; #4自检-HMI
OUT W29.11  ; #4左右自检气缸自检缩回
; rung 14: 手动异常提示    左自检气缸
@LD W6.07  ; 自检左气缸-HMI
@OR W6.11  ; 左夹爪气缸-HMI
ANDNOT T0048  ; #4左密封气缸缩回位时间
OR 106.12  ; #4左密封气缸没缩回异常
ANDNOT T0272  ; #4左密封气缸没缩回异常提示持续时间
OUT 106.12  ; #4左密封气缸没缩回异常
TIMX(550) 0272 &50  ; #4左密封气缸没缩回异常提示持续时间
; rung 15: 右自检气缸异常
@LD W6.08  ; 自检右气缸-HMI
@OR W6.12  ; 右夹爪气缸-HMI
ANDNOT T0050  ; #4右密封气缸缩回位时间
OR 106.13  ; #4右密封气缸没缩回异常
ANDNOT T0273  ; #4右密封气缸没缩回异常
OUT 106.13  ; #4右密封气缸没缩回异常
TIMX(550) 0273 &50  ; #4右密封气缸没缩回异常
; rung 16
ILC(003)

### Section 模组_1自动

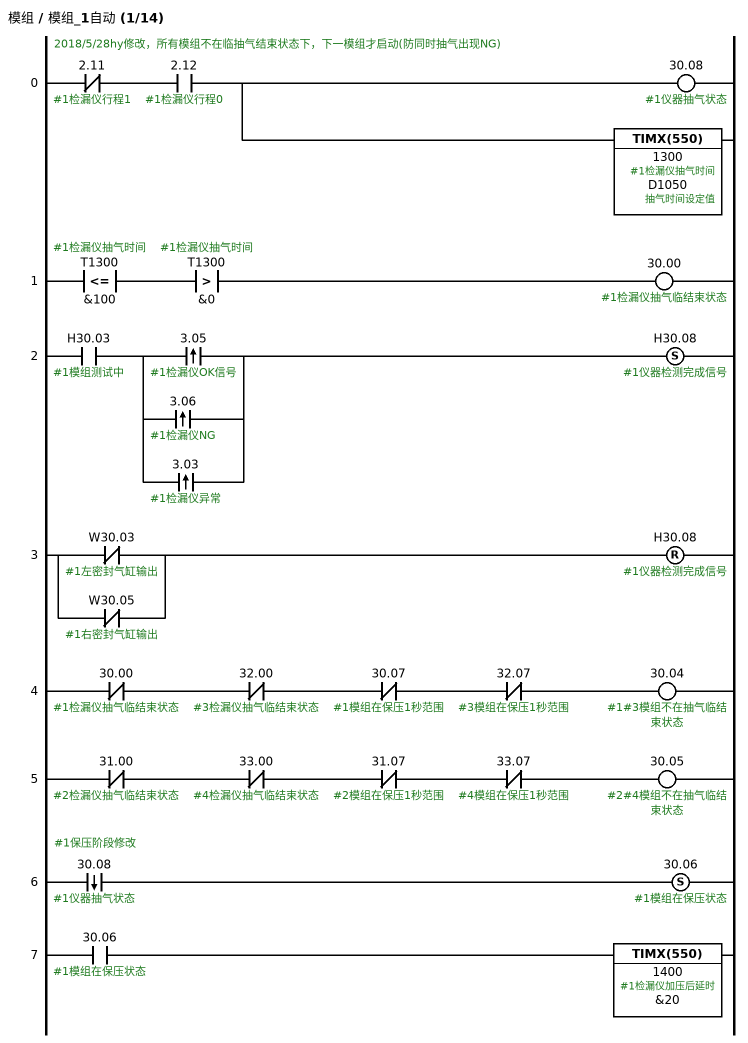
; rung 0: 2018/5/28hy修改，所有模组不在临抽气结束状态下，下一模组才启动(防同时抽气出现NG)
LDNOT 2.11  ; #1检漏仪行程1
AND 2.12  ; #1检漏仪行程0
OUT 30.08  ; #1仪器抽气状态
TIMX(550) 1300 D1050  ; 抽气时间设定值, #1检漏仪抽气时间
; rung 1
LD<=(315) T1300 &100  ; #1检漏仪抽气时间
AND>(320) T1300 &0  ; #1检漏仪抽气时间
OUT 30.00  ; #1检漏仪抽气临结束状态
; rung 2
LD H30.03  ; #1模组测试中
@LD 3.05  ; #1检漏仪OK信号
@OR 3.06  ; #1检漏仪NG
@OR 3.03  ; #1检漏仪异常
ANDLD
SET H30.08  ; #1仪器检测完成信号
; rung 3
LDNOT W30.03  ; #1左密封气缸输出
ORNOT W30.05  ; #1右密封气缸输出
RSET H30.08  ; #1仪器检测完成信号
; rung 4
LDNOT 30.00  ; #1检漏仪抽气临结束状态
ANDNOT 32.00  ; #3检漏仪抽气临结束状态
ANDNOT 30.07  ; #1模组在保压1秒范围
ANDNOT 32.07  ; #3模组在保压1秒范围
OUT 30.04  ; #1#3模组不在抽气临结束状态
; rung 5
LDNOT 31.00  ; #2检漏仪抽气临结束状态
ANDNOT 33.00  ; #4检漏仪抽气临结束状态
ANDNOT 31.07  ; #2模组在保压1秒范围
ANDNOT 33.07  ; #4模组在保压1秒范围
OUT 30.05  ; #2#4模组不在抽气临结束状态
; rung 6: #1保压阶段修改
%LD 30.08  ; #1仪器抽气状态
SET 30.06  ; #1模组在保压状态
; rung 7
LD 30.06  ; #1模组在保压状态
TIMX(550) 1400 &20  ; #1检漏仪加压后延时

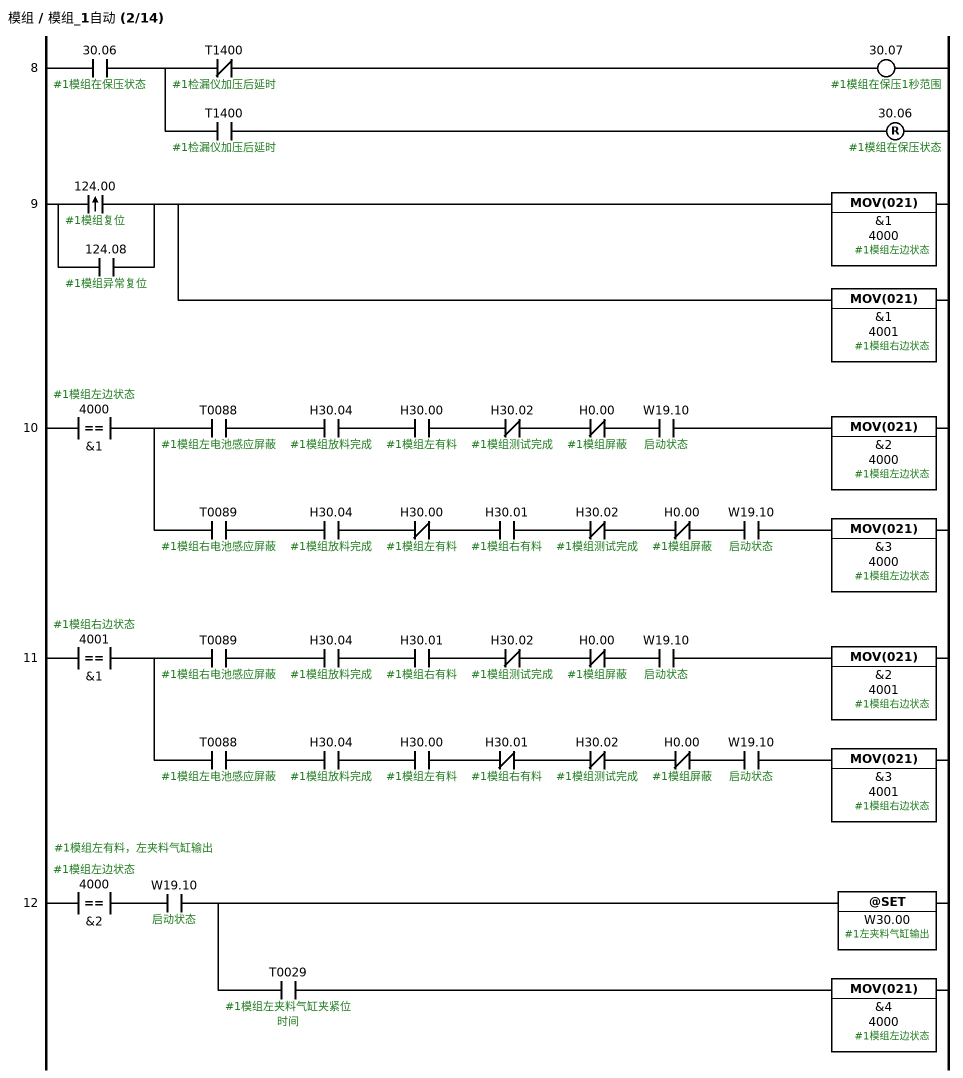
; rung 8
LD 30.06  ; #1模组在保压状态
OUT TR0
ANDNOT T1400  ; #1检漏仪加压后延时
OUT 30.07  ; #1模组在保压1秒范围
LD TR0
AND T1400  ; #1检漏仪加压后延时
RSET 30.06  ; #1模组在保压状态
; rung 9
@LD 124.00  ; #1模组复位
OR 124.08  ; #1模组异常复位
MOV(021) &1 4000  ; #1模组左边状态
MOV(021) &1 4001  ; #1模组右边状态
; rung 10
LD=(300) 4000 &1  ; #1模组左边状态
OUT TR0
AND T0088  ; #1模组左电池感应屏蔽
AND H30.04  ; #1模组放料完成
AND H30.00  ; #1模组左有料
ANDNOT H30.02  ; #1模组测试完成
ANDNOT H0.00  ; #1模组屏蔽
AND W19.10  ; 启动状态
MOV(021) &2 4000  ; #1模组左边状态
LD TR0
AND T0089  ; #1模组右电池感应屏蔽
AND H30.04  ; #1模组放料完成
ANDNOT H30.00  ; #1模组左有料
AND H30.01  ; #1模组右有料
ANDNOT H30.02  ; #1模组测试完成
ANDNOT H0.00  ; #1模组屏蔽
AND W19.10  ; 启动状态
MOV(021) &3 4000  ; #1模组左边状态
; rung 11
LD=(300) 4001 &1  ; #1模组右边状态
OUT TR0
AND T0089  ; #1模组右电池感应屏蔽
AND H30.04  ; #1模组放料完成
AND H30.01  ; #1模组右有料
ANDNOT H30.02  ; #1模组测试完成
ANDNOT H0.00  ; #1模组屏蔽
AND W19.10  ; 启动状态
MOV(021) &2 4001  ; #1模组右边状态
LD TR0
AND T0088  ; #1模组左电池感应屏蔽
AND H30.04  ; #1模组放料完成
AND H30.00  ; #1模组左有料
ANDNOT H30.01  ; #1模组右有料
ANDNOT H30.02  ; #1模组测试完成
ANDNOT H0.00  ; #1模组屏蔽
AND W19.10  ; 启动状态
MOV(021) &3 4001  ; #1模组右边状态
; rung 12: #1模组左有料，左夹料气缸输出
LD=(300) 4000 &2  ; #1模组左边状态
AND W19.10  ; 启动状态
@SET W30.00  ; #1左夹料气缸输出
AND T0029  ; #1模组左夹料气缸夹紧位时间
MOV(021) &4 4000  ; #1模组左边状态

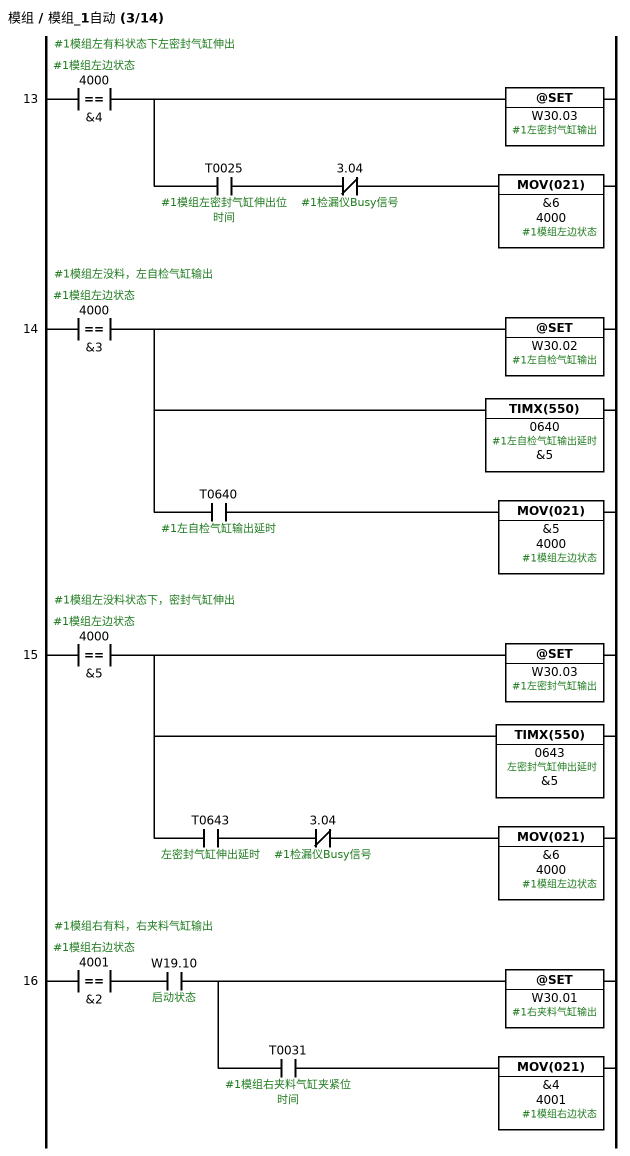
; rung 13: #1模组左有料状态下左密封气缸伸出
LD=(300) 4000 &4  ; #1模组左边状态
@SET W30.03  ; #1左密封气缸输出
AND T0025  ; #1模组左密封气缸伸出位时间
ANDNOT 3.04  ; #1检漏仪Busy信号
MOV(021) &6 4000  ; #1模组左边状态
; rung 14: #1模组左没料，左自检气缸输出
LD=(300) 4000 &3  ; #1模组左边状态
@SET W30.02  ; #1左自检气缸输出
TIMX(550) 0640 &5  ; #1左自检气缸输出延时
AND T0640  ; #1左自检气缸输出延时
MOV(021) &5 4000  ; #1模组左边状态
; rung 15: #1模组左没料状态下，密封气缸伸出
LD=(300) 4000 &5  ; #1模组左边状态
@SET W30.03  ; #1左密封气缸输出
TIMX(550) 0643 &5  ; 左密封气缸伸出延时
AND T0643  ; 左密封气缸伸出延时
ANDNOT 3.04  ; #1检漏仪Busy信号
MOV(021) &6 4000  ; #1模组左边状态
; rung 16: #1模组右有料，右夹料气缸输出
LD=(300) 4001 &2  ; #1模组右边状态
AND W19.10  ; 启动状态
@SET W30.01  ; #1右夹料气缸输出
AND T0031  ; #1模组右夹料气缸夹紧位时间
MOV(021) &4 4001  ; #1模组右边状态

